FUNCTION_BLOCK AX_FB_F_TRIG (* Detect falling edge with AX Adapter *)
  (* Standard: 61499-1; Description: Copyright (c) 2023 Martin Erich Jobst, HR Agrartechnik GmbH This program and the accompanying materials are made available under the terms of the Eclipse Public License 2.0 which is available at https://www.eclipse.org/legal/epl-2.0/ SPDX-License-Identifier: EPL-2.0 *)
  (* Version 3.0, 2025-02-01, Franz Höpfinger, AX version *)
  (* Version 1.0, 2023-04-28, Martin Jobst, initial API and implementation and/or initial documentation *)
  PACKAGE adapter::iec61131::edgeDetection;
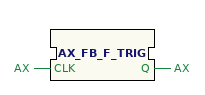
  SOCKETS
    CLK : adapter::types::unidirectional::AX; (* Clock *)
  END_SOCKETS
  PLUGS
    Q : adapter::types::unidirectional::AX; (* Output *)
  END_PLUGS
  VAR
    MEM : BOOL := TRUE;
  END_VAR
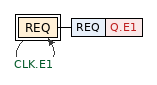
  EC_STATES
    REQ : REQ -> Q.E1;
  END_STATES
  EC_TRANSITIONS
    REQ TO REQ := CLK.E1;
  END_TRANSITIONS
  ALGORITHM REQ IN ST:
Q.D1 := NOT CLK.D1 AND NOT MEM;
MEM := NOT CLK.D1;
  END_ALGORITHM
END_FUNCTION_BLOCK
